(* Logix 5000 project; controller FRIST_EXAMPLE Emulate 5570 rev 19.11; software revision 19.01 *)

TASK MainTask (continuous, watchdog 500 ms) : MainProgram

MODULES
   Local : Emulate 5570 (ICP 2, rev 19.11)
       : 1756-IB32 (ICP 3, rev 3.1, Input RPI 20 ms)   // DG-INPUT
       : vendor 1 type 7 code 8 (ICP 4, rev 3.1, Output RPI 20 ms)
       : 1756-IF6I (ICP 5, rev 1.1, Input RPI 100 ms)
       : 1756-OF8 (ICP 6, rev 1.1, Output RPI 12 ms)
END_MODULES

VAR_GLOBAL   (* controller tags *)
   LIGA : BOOL;
END_VAR

PROGRAM MainProgram   (* main routine MainRoutine *)
VAR
   PARAM1 : DINT := 5;
   PARAM2 : DINT := 4;
   RESULTADO : DINT := 9;
   VAR1 : DINT := 5;
   VAR2 : DINT := 4;
   VAR_RESULTADO : DINT := 9;
END_VAR

ROUTINE CALCULAR   (* ladder *)
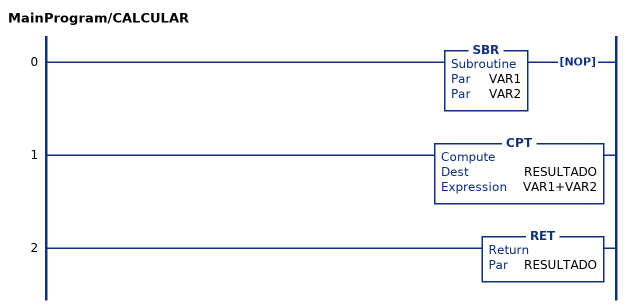
   0: SBR(VAR1,VAR2)NOP();
   1: CPT(RESULTADO,VAR1+VAR2);
   2: RET(RESULTADO);
END_ROUTINE

ROUTINE MainRoutine   (* ladder *)
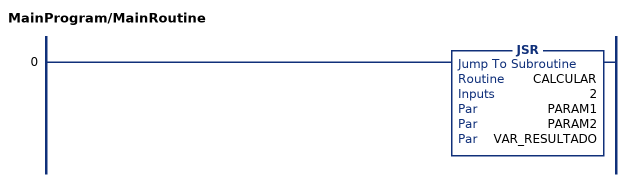
   0: JSR(CALCULAR,2,PARAM1,PARAM2,VAR_RESULTADO);
END_ROUTINE
END_PROGRAM
